FUNCTION_BLOCK Mediator
VAR_INPUT

	MoverArray		: ARRAY [0..GVL.NUM_MOVERS-1] OF POINTER TO Mover;
	StationArray	: ARRAY [0..GVL.NUM_MOVERS-1] OF POINTER TO Station;

END_VAR
VAR_OUTPUT
END_VAR
VAR
END_VAR

END_FUNCTION_BLOCK

(* stored: Version 1.1.0.1, ProductVersion 3.1.4024.12
   POU Mediator: Id {164d51b4-07ec-0e46-0eb0-392af39d7d3a}, SpecialFunc None *)
